FUNCTION_BLOCK FailScenarioHMI (* Composite Function Block Type *)
  (* Standard: 61499-2 *)
  (* Version 0.0, 5/14/2019, erik, nxtControl GmbH, template *)
  PACKAGE Main;
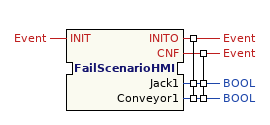
  EVENT_INPUT
    INIT; (* Initialization Request *)
  END_EVENT
  EVENT_OUTPUT
    INITO WITH Jack1, Conveyor1; (* Initialization Confirm *)
    CNF WITH Jack1, Conveyor1; (* Execution Confirmation *)
  END_EVENT
  VAR_OUTPUT
    Jack1 : BOOL; (* Output event qualifier *)
    Conveyor1 : BOOL;
  END_VAR
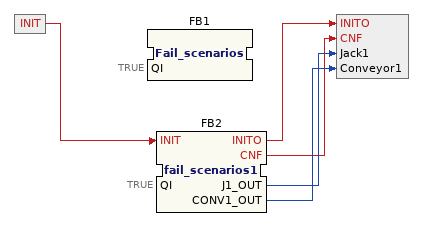
  FBS
    FB1 : Fail_scenarios(QI := TRUE);
    FB2 : fail_scenarios1(QI := TRUE);
  END_FBS
  EVENT_CONNECTIONS
    INIT TO FB2.INIT;
    FB2.INITO TO INITO;
    FB2.CNF TO CNF;
  END_CONNECTIONS
  DATA_CONNECTIONS
    FB2.J1_OUT TO Jack1;
    FB2.CONV1_OUT TO Conveyor1;
  END_CONNECTIONS
END_FUNCTION_BLOCK
